(* Logix 5000 project; controller cal1615 1756-L62 rev 20.19; software revision 20.05; part 25 of 81 *)
(* tags used below, declared in another part *)
   FAULT : BOOL;   // Fault AFI
   p01_param_oven_timer_presets : DINT[32];   // System Parameter Oven Timer Presets
   p01_param_process_air_hl : REAL;   // Machine Parameter Process Air High Limit
   p01_sys_lc : Limit_Clamp;   // Zone 1 Misc Control Limit Clamp
   p01r09_pb_global_reset : BOOL;   // System Modes PB: Global Fault Reset
   p01r11 : routine;   // System Timer Presets
   p02_real_from_hmi : hmi_real;   // MOP HMI Iface Real from HMI
   p12_dint_to_hmi : DINT[16];   // Zone 2 Temperature Control VFDs On
   p12_param_fast_to_soak : REAL;   // Zone 2 Parameter Fast to Soak Control
   p12_param_lfl_hhl : REAL;   // Zone 2 Parameter High High Lower Flash Limit
   p12_param_lfl_hl : REAL;   // Zone 2 Parameter High LFL Limit
   p12_param_pid1_ff : REAL;   // Zone 2 Parameter Fast PID Bias
   p12_param_pid1_kd : REAL;   // Zone 2 Parameter Fast PID Derivative Gain
   p12_param_pid1_ki : REAL;   // Zone 2 Parameter Fast PID Integral Gain
   p12_param_pid1_kp : REAL;   // Zone 2 Parameter Fast PID Proportional Gain
   p12_param_pid2_ff : REAL;   // Zone 2 Parameter Auto PID Bias
   p12_param_pid2_kd : REAL;   // Zone 2 Parameter Auto PID Derivative Gain
   p12_param_pid2_ki : REAL;   // Zone 2 Parameter Auto PID Integral Gain
   p12_param_pid2_kp : REAL;   // Zone 2 Parameter Auto PID Proportional Gain
   p12_param_shutdown_temp : REAL;   // Zone 2 Parameter Zone Shutdown Temperature
   p12_param_soak_to_fast : REAL;   // Zone 2 Parameter Soak to Fast Control
   p12_param_tc01_dev : REAL;   // Zone 2 Parameter Oven Temperature Deviation from Setpoint
   p12_param_tc01_hl : REAL;   // Zone 2 Parameter Process Air High Limit
   p12_param_tc01z : REAL;   // Zone 2 Parameter Process Temperature Zero Offset
   p12_param_tc02z : REAL;   // Zone 2 Parameter SupplyTemperature Zero Offset
   p12_param_zone_pressure : REAL;   // Zone 2 Parameter High Pressure LImit
   p12r01 : routine;   // Zone 2 Main
   p12r02 : routine;   // Zone 2 Misc Control
   p12r02_timer_safe_temp : TIMER[2];   // Zone 2 Misc Control Chamber SafeTemperature Dwell
   p12r02_timer_warning : TIMER[4];   // Zone 2 Misc Control Warning Delay
   p12r08 : routine;   // Zone 2 Warnings
   p12r08_timer_fault : TIMER[4];   // Zone 2 Warnings Fault Delay
   p12r08_timer_warning : TIMER[4];   // Zone 2 Warnings Warning Delay
   p12r09 : routine;   // Zone 2 Modes
   p12r09_timer_fault : TIMER[4];   // Zone 2 Modes Fault Delay
   p12r09_timer_warning : TIMER[8];   // Zone 2 Modes Warning Delay
   p12r10 : routine;   // Zone 2
   p12r10_timer_fault : TIMER[4];   // Zone 2 Fault Delay
   p12r10_timer_warning : TIMER[4];   // Zone 2 Warning Delay
   p12r20_timer_state_11 : TIMER;   // Zone 2 Temp Sequence State 11 Dwell
   p12r20_timer_state_3 : TIMER;   // Zone 2 Temperature Control State 3 Dwell
   p12r20_timer_state_4 : TIMER;   // Zone 2 Temp Sequence State 4 Dwell
   p12r20_timer_state_7 : TIMER;   // Zone 2 Temp Sequence State 7 Dwell
   p12r30 : routine;   // Zone 2 Temperature Control
   p12r30_cv_man_sp : REAL;   // Zone 2 Temperature Control Manual Heat Control Valve Setpoint
   p12r30_temp_deviation_setpoint : DINT;
   p12r30_timer_fault : TIMER[16];   // Zone 2 Temperature Control Fault Delay
   p12r30_timer_warning : TIMER[12];   // Zone 2 Temperature Control Warning Delay
   p12r31 : routine;   // Zone 2 Exhaust VFD
   p12r31_timer_fault : TIMER[5];   // Zone 2 Exhaust VFD Fault Timer
   p12r31_timer_warning : TIMER[5];   // Zone 2 Exhaust VFD Waringing Timer
   p12r32 : routine;   // Zone 2 Recirc VFD
   p12r32_timer_fault : TIMER[5];   // Zone 2 Recirc VFD Fault Timer
   p12r32_timer_warning : TIMER[5];   // Zone 2 Supply VFD Warning Timer
(* P12_Zone_2, continued *)

ROUTINE R08_Warnings   (* ladder *)
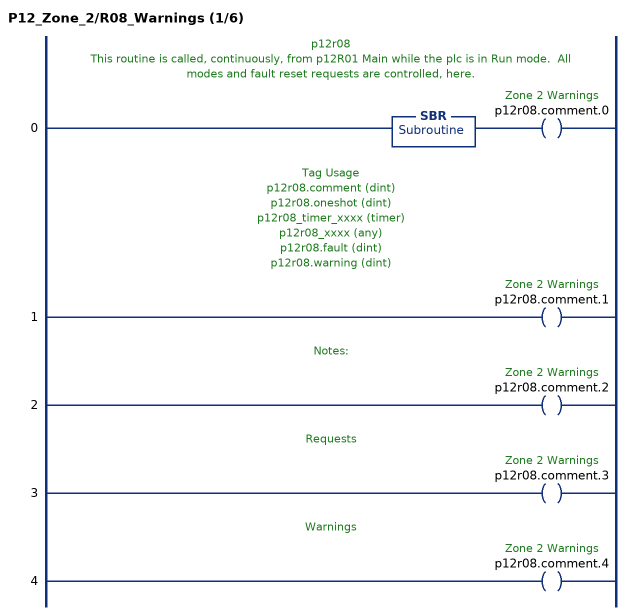
   // p12r08
   // This routine is called, continuously, from p12R01 Main while the plc is in Run mode.  All modes and fault reset requests are controlled, here.
   0: SBR()OTE(p12r08.comment.0);
   // Tag Usage
   // p12r08.comment (dint)
   // p12r08.oneshot (dint)
   // p12r08_timer_xxxx (timer)
   // p12r08_xxxx (any)
   // p12r08.fault (dint)
   // p12r08.warning (dint)
   1: OTE(p12r08.comment.1);
   // Notes:
   2: OTE(p12r08.comment.2);
   // Requests
   3: OTE(p12r08.comment.3);
   // Warnings
   4: OTE(p12r08.comment.4);
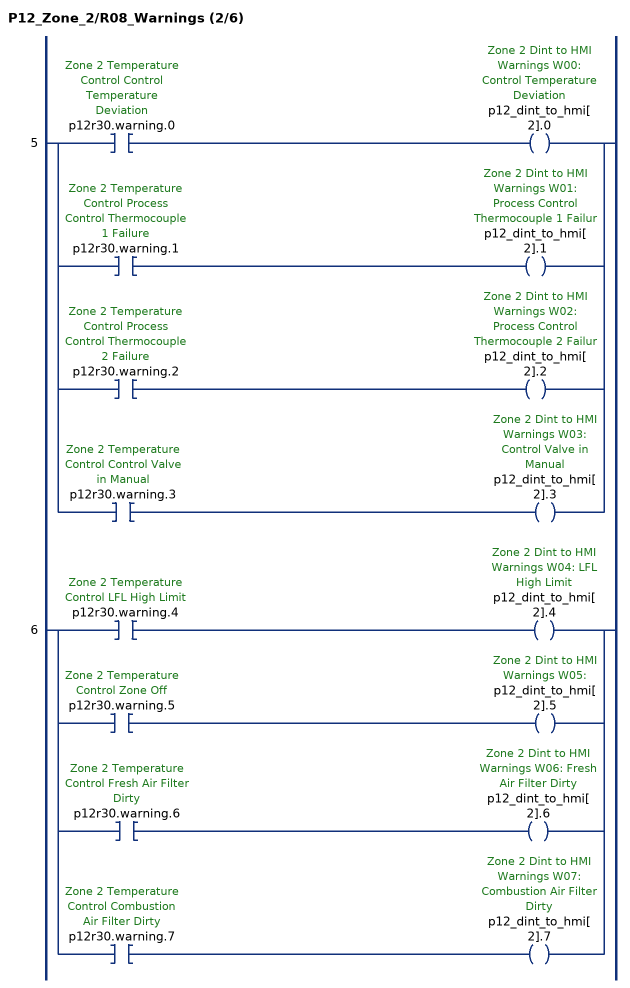
   5: [XIC(p12r30.warning.0) OTE(p12_dint_to_hmi[2].0) ,XIC(p12r30.warning.1) OTE(p12_dint_to_hmi[2].1) ,XIC(p12r30.warning.2) OTE(p12_dint_to_hmi[2].2) ,XIC(p12r30.warning.3) OTE(p12_dint_to_hmi[2].3) ];
   6: [XIC(p12r30.warning.4) OTE(p12_dint_to_hmi[2].4) ,XIC(p12r30.warning.5) OTE(p12_dint_to_hmi[2].5) ,XIC(p12r30.warning.6) OTE(p12_dint_to_hmi[2].6) ,XIC(p12r30.warning.7) OTE(p12_dint_to_hmi[2].7) ];
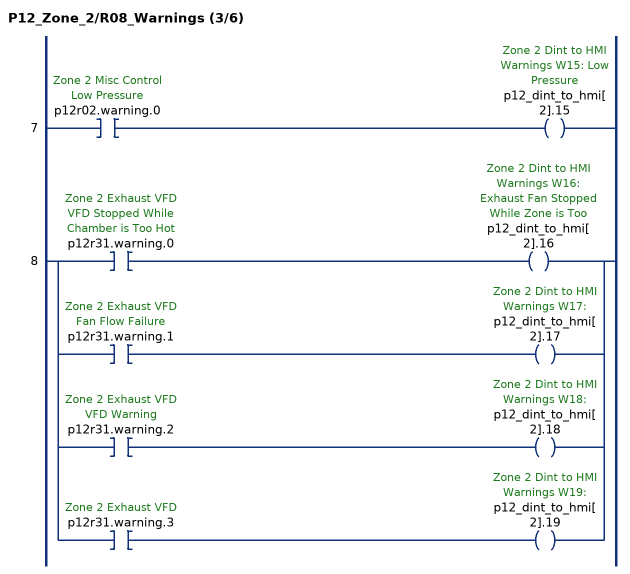
   7: XIC(p12r02.warning.0)OTE(p12_dint_to_hmi[2].15);
   8: [XIC(p12r31.warning.0) OTE(p12_dint_to_hmi[2].16) ,XIC(p12r31.warning.1) OTE(p12_dint_to_hmi[2].17) ,XIC(p12r31.warning.2) OTE(p12_dint_to_hmi[2].18) ,XIC(p12r31.warning.3) OTE(p12_dint_to_hmi[2].19) ];
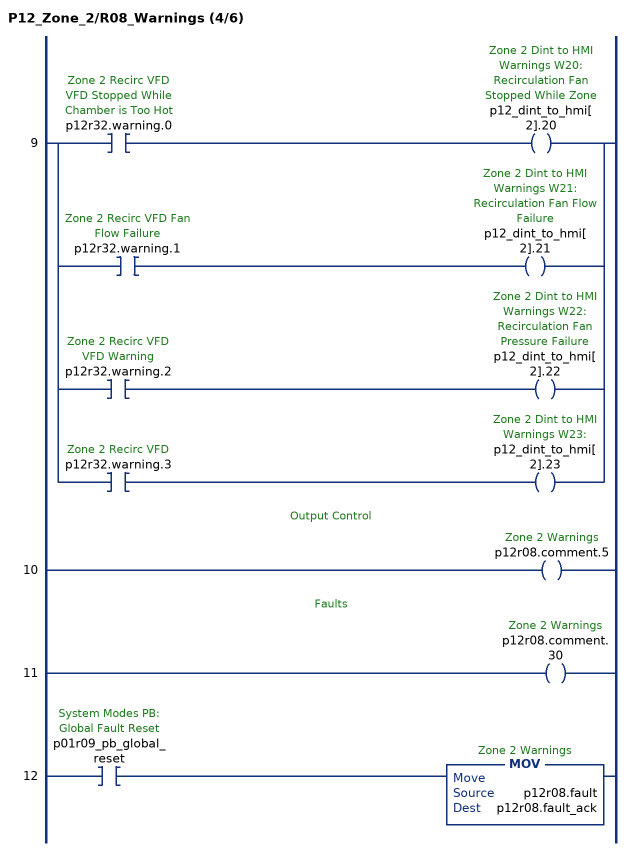
   9: [XIC(p12r32.warning.0) OTE(p12_dint_to_hmi[2].20) ,XIC(p12r32.warning.1) OTE(p12_dint_to_hmi[2].21) ,XIC(p12r32.warning.2) OTE(p12_dint_to_hmi[2].22) ,XIC(p12r32.warning.3) OTE(p12_dint_to_hmi[2].23) ];
   // Output Control
   10: OTE(p12r08.comment.5);
   // Faults
   11: OTE(p12r08.comment.30);
   12: XIC(p01r09_pb_global_reset)MOV(p12r08.fault,p12r08.fault_ack);
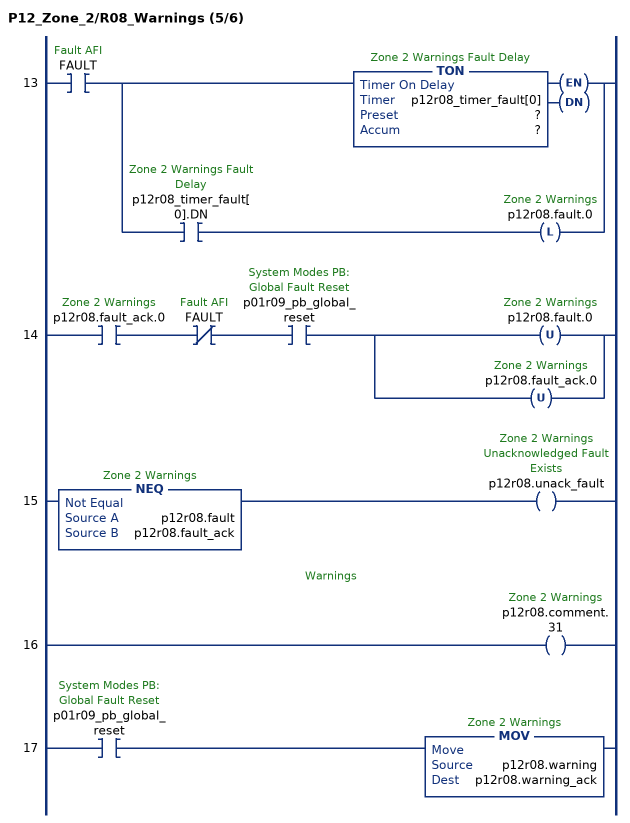
   13: XIC(FAULT)[TON(p12r08_timer_fault[0],?,?) ,XIC(p12r08_timer_fault[0].DN) OTL(p12r08.fault.0) ];
   14: XIC(p12r08.fault_ack.0)XIO(FAULT)XIC(p01r09_pb_global_reset)[OTU(p12r08.fault.0) ,OTU(p12r08.fault_ack.0) ];
   15: NEQ(p12r08.fault,p12r08.fault_ack)OTE(p12r08.unack_fault);
   // Warnings
   16: OTE(p12r08.comment.31);
   17: XIC(p01r09_pb_global_reset)MOV(p12r08.warning,p12r08.warning_ack);
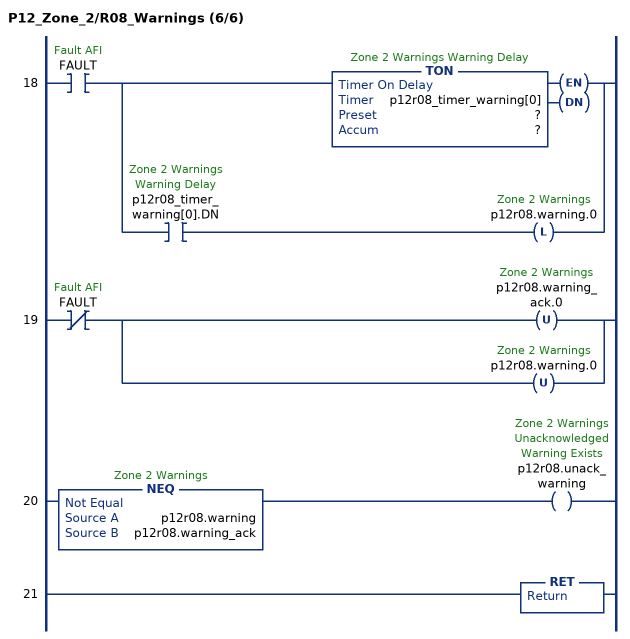
   18: XIC(FAULT)[TON(p12r08_timer_warning[0],?,?) ,XIC(p12r08_timer_warning[0].DN) OTL(p12r08.warning.0) ];
   19: XIO(FAULT)[OTU(p12r08.warning_ack.0) ,OTU(p12r08.warning.0) ];
   20: NEQ(p12r08.warning,p12r08.warning_ack)OTE(p12r08.unack_warning);
   21: RET();
END_ROUTINE

ROUTINE R09_Modes   (* ladder *)
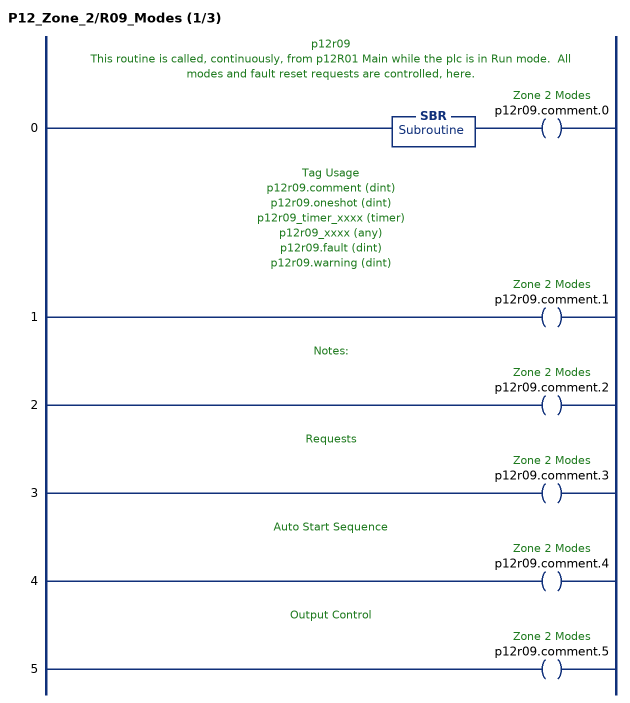
   // p12r09
   // This routine is called, continuously, from p12R01 Main while the plc is in Run mode.  All modes and fault reset requests are controlled, here.
   0: SBR()OTE(p12r09.comment.0);
   // Tag Usage
   // p12r09.comment (dint)
   // p12r09.oneshot (dint)
   // p12r09_timer_xxxx (timer)
   // p12r09_xxxx (any)
   // p12r09.fault (dint)
   // p12r09.warning (dint)
   1: OTE(p12r09.comment.1);
   // Notes:
   2: OTE(p12r09.comment.2);
   // Requests
   3: OTE(p12r09.comment.3);
   // Auto Start Sequence
   4: OTE(p12r09.comment.4);
   // Output Control
   5: OTE(p12r09.comment.5);
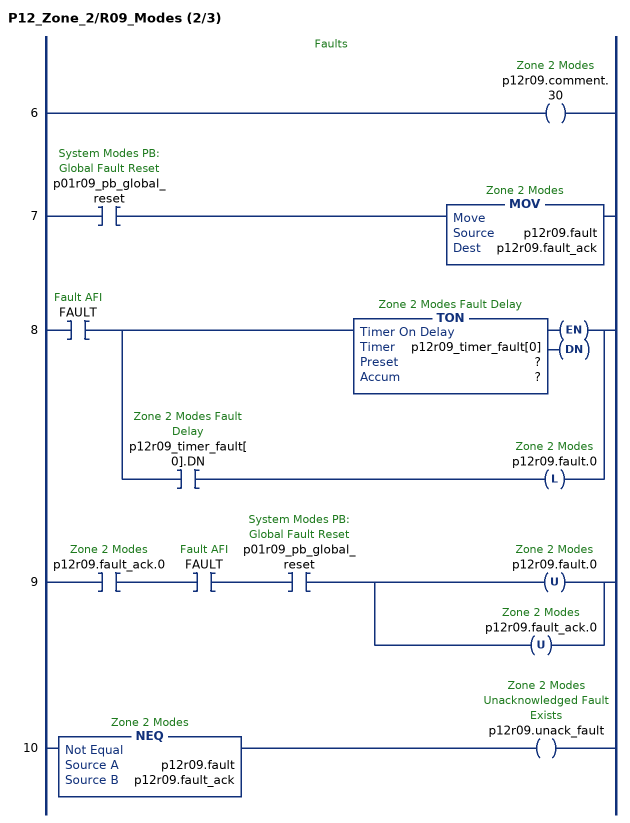
   // Faults
   6: OTE(p12r09.comment.30);
   7: XIC(p01r09_pb_global_reset)MOV(p12r09.fault,p12r09.fault_ack);
   8: XIC(FAULT)[TON(p12r09_timer_fault[0],?,?) ,XIC(p12r09_timer_fault[0].DN) OTL(p12r09.fault.0) ];
   9: XIC(p12r09.fault_ack.0)XIC(FAULT)XIC(p01r09_pb_global_reset)[OTU(p12r09.fault.0) ,OTU(p12r09.fault_ack.0) ];
   10: NEQ(p12r09.fault,p12r09.fault_ack)OTE(p12r09.unack_fault);
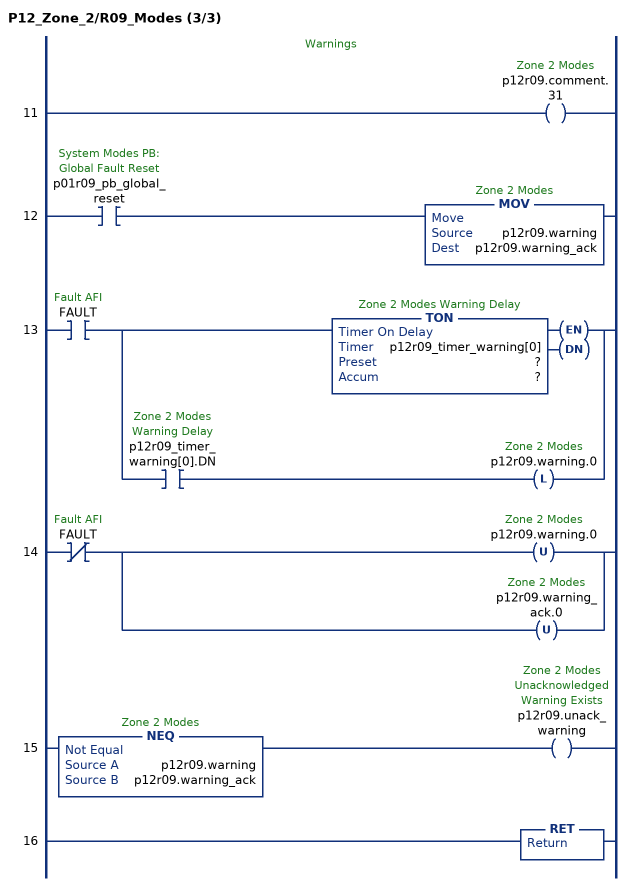
   // Warnings
   11: OTE(p12r09.comment.31);
   12: XIC(p01r09_pb_global_reset)MOV(p12r09.warning,p12r09.warning_ack);
   13: XIC(FAULT)[TON(p12r09_timer_warning[0],?,?) ,XIC(p12r09_timer_warning[0].DN) OTL(p12r09.warning.0) ];
   14: XIO(FAULT)[OTU(p12r09.warning.0) ,OTU(p12r09.warning_ack.0) ];
   15: NEQ(p12r09.warning,p12r09.warning_ack)OTE(p12r09.unack_warning);
   16: RET();
END_ROUTINE

ROUTINE R10_Parameters   (* ladder *)
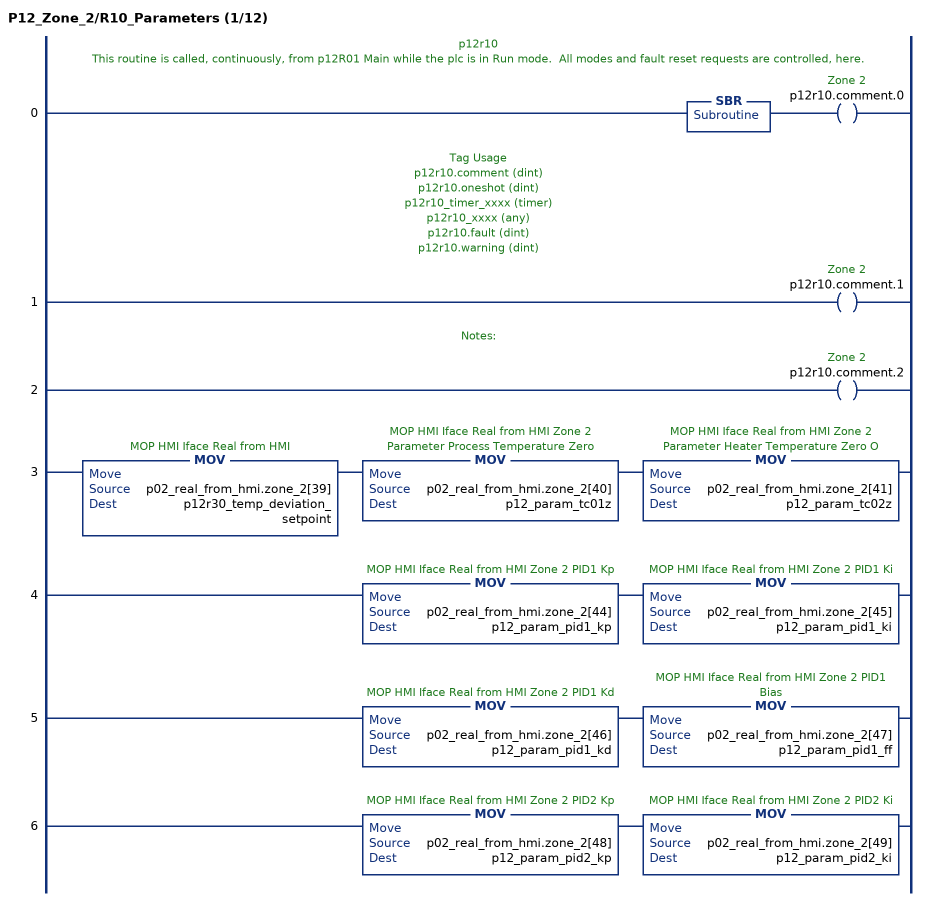
   // p12r10
   // This routine is called, continuously, from p12R01 Main while the plc is in Run mode.  All modes and fault reset requests are controlled, here.
   0: SBR()OTE(p12r10.comment.0);
   // Tag Usage
   // p12r10.comment (dint)
   // p12r10.oneshot (dint)
   // p12r10_timer_xxxx (timer)
   // p12r10_xxxx (any)
   // p12r10.fault (dint)
   // p12r10.warning (dint)
   1: OTE(p12r10.comment.1);
   // Notes:
   2: OTE(p12r10.comment.2);
   3: MOV(p02_real_from_hmi.zone_2[39],p12r30_temp_deviation_setpoint)MOV(p02_real_from_hmi.zone_2[40],p12_param_tc01z)MOV(p02_real_from_hmi.zone_2[41],p12_param_tc02z);
   4: MOV(p02_real_from_hmi.zone_2[44],p12_param_pid1_kp)MOV(p02_real_from_hmi.zone_2[45],p12_param_pid1_ki);
   5: MOV(p02_real_from_hmi.zone_2[46],p12_param_pid1_kd)MOV(p02_real_from_hmi.zone_2[47],p12_param_pid1_ff);
   6: MOV(p02_real_from_hmi.zone_2[48],p12_param_pid2_kp)MOV(p02_real_from_hmi.zone_2[49],p12_param_pid2_ki);
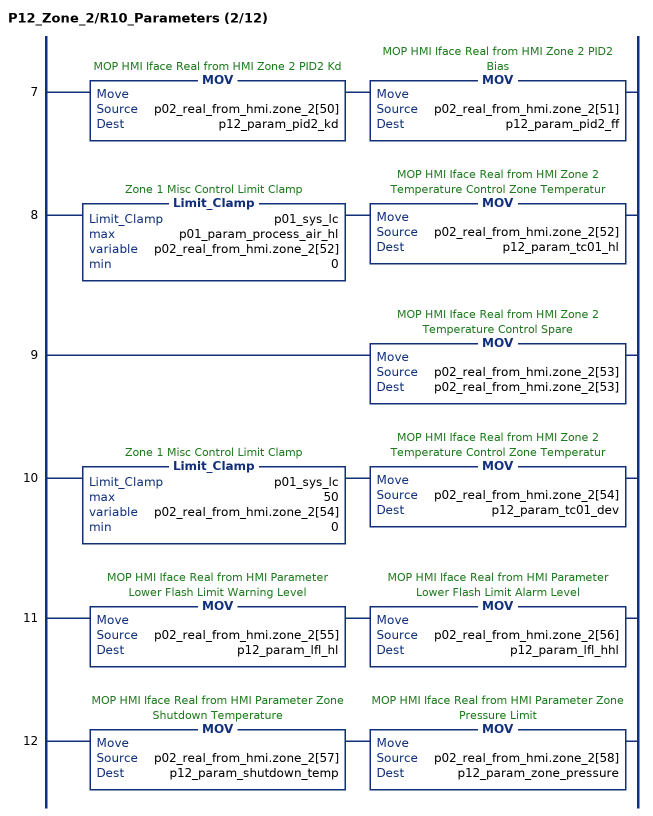
   7: MOV(p02_real_from_hmi.zone_2[50],p12_param_pid2_kd)MOV(p02_real_from_hmi.zone_2[51],p12_param_pid2_ff);
   8: Limit_Clamp(p01_sys_lc,p01_param_process_air_hl,p02_real_from_hmi.zone_2[52],0)MOV(p02_real_from_hmi.zone_2[52],p12_param_tc01_hl);
   9: MOV(p02_real_from_hmi.zone_2[53],p02_real_from_hmi.zone_2[53]);
   10: Limit_Clamp(p01_sys_lc,50,p02_real_from_hmi.zone_2[54],0)MOV(p02_real_from_hmi.zone_2[54],p12_param_tc01_dev);
   11: MOV(p02_real_from_hmi.zone_2[55],p12_param_lfl_hl)MOV(p02_real_from_hmi.zone_2[56],p12_param_lfl_hhl);
   12: MOV(p02_real_from_hmi.zone_2[57],p12_param_shutdown_temp)MOV(p02_real_from_hmi.zone_2[58],p12_param_zone_pressure);
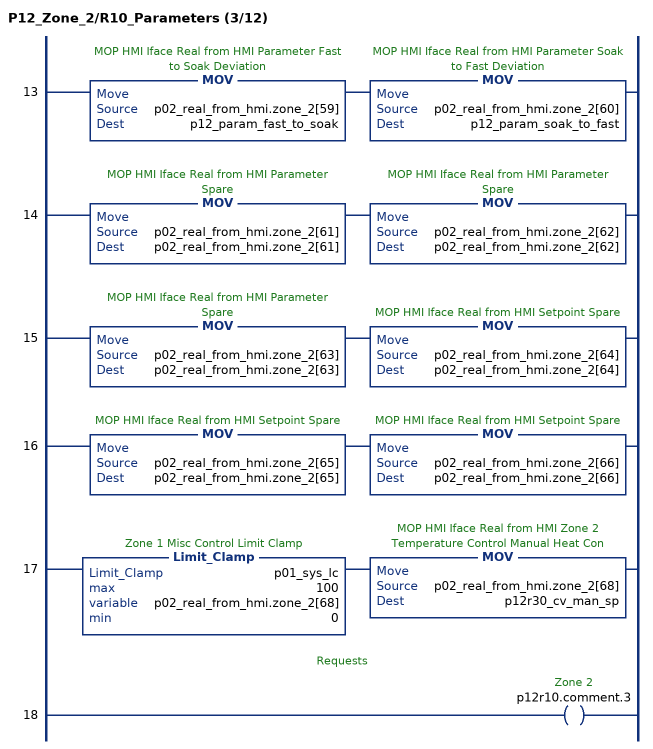
   13: MOV(p02_real_from_hmi.zone_2[59],p12_param_fast_to_soak)MOV(p02_real_from_hmi.zone_2[60],p12_param_soak_to_fast);
   14: MOV(p02_real_from_hmi.zone_2[61],p02_real_from_hmi.zone_2[61])MOV(p02_real_from_hmi.zone_2[62],p02_real_from_hmi.zone_2[62]);
   15: MOV(p02_real_from_hmi.zone_2[63],p02_real_from_hmi.zone_2[63])MOV(p02_real_from_hmi.zone_2[64],p02_real_from_hmi.zone_2[64]);
   16: MOV(p02_real_from_hmi.zone_2[65],p02_real_from_hmi.zone_2[65])MOV(p02_real_from_hmi.zone_2[66],p02_real_from_hmi.zone_2[66]);
   17: Limit_Clamp(p01_sys_lc,100,p02_real_from_hmi.zone_2[68],0)MOV(p02_real_from_hmi.zone_2[68],p12r30_cv_man_sp);
   // Requests
   18: OTE(p12r10.comment.3);
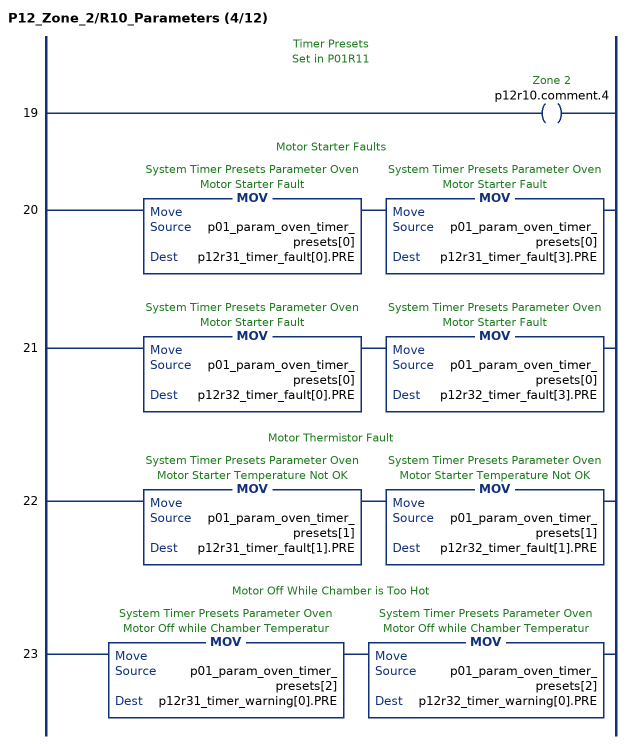
   // Timer Presets
   // Set in P01R11
   19: OTE(p12r10.comment.4);
   // Motor Starter Faults
   20: MOV(p01_param_oven_timer_presets[0],p12r31_timer_fault[0].PRE)MOV(p01_param_oven_timer_presets[0],p12r31_timer_fault[3].PRE);
   21: MOV(p01_param_oven_timer_presets[0],p12r32_timer_fault[0].PRE)MOV(p01_param_oven_timer_presets[0],p12r32_timer_fault[3].PRE);
   // Motor Thermistor Fault
   22: MOV(p01_param_oven_timer_presets[1],p12r31_timer_fault[1].PRE)MOV(p01_param_oven_timer_presets[1],p12r32_timer_fault[1].PRE);
   // Motor Off While Chamber is Too Hot
   23: MOV(p01_param_oven_timer_presets[2],p12r31_timer_warning[0].PRE)MOV(p01_param_oven_timer_presets[2],p12r32_timer_warning[0].PRE);
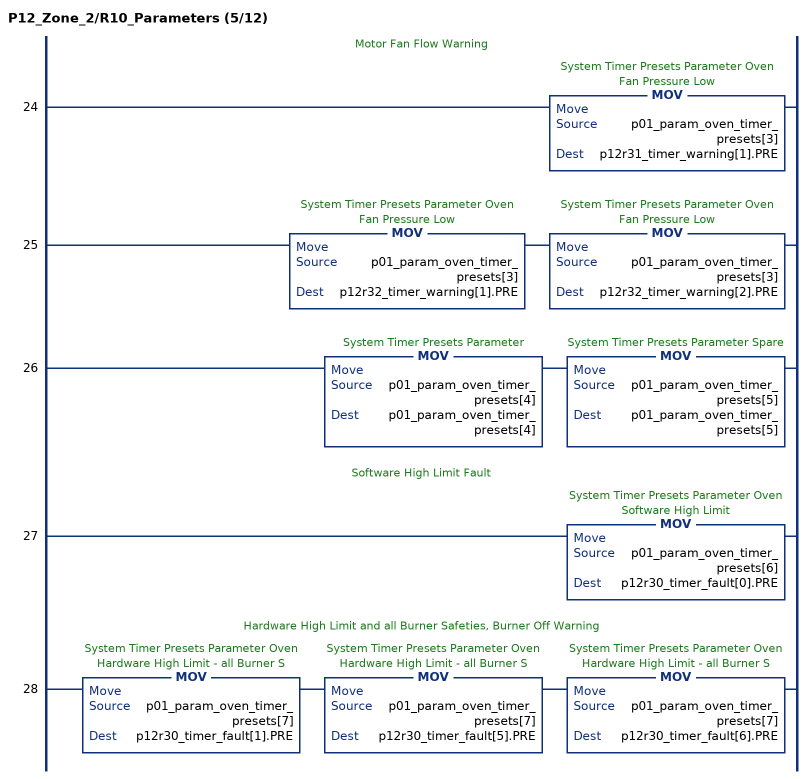
   // Motor Fan Flow Warning
   24: MOV(p01_param_oven_timer_presets[3],p12r31_timer_warning[1].PRE);
   25: MOV(p01_param_oven_timer_presets[3],p12r32_timer_warning[1].PRE)MOV(p01_param_oven_timer_presets[3],p12r32_timer_warning[2].PRE);
   26: MOV(p01_param_oven_timer_presets[4],p01_param_oven_timer_presets[4])MOV(p01_param_oven_timer_presets[5],p01_param_oven_timer_presets[5]);
   // Software High Limit Fault
   27: MOV(p01_param_oven_timer_presets[6],p12r30_timer_fault[0].PRE);
   // Hardware High Limit and all Burner Safeties, Burner Off Warning
   28: MOV(p01_param_oven_timer_presets[7],p12r30_timer_fault[1].PRE)MOV(p01_param_oven_timer_presets[7],p12r30_timer_fault[5].PRE)MOV(p01_param_oven_timer_presets[7],p12r30_timer_fault[6].PRE);
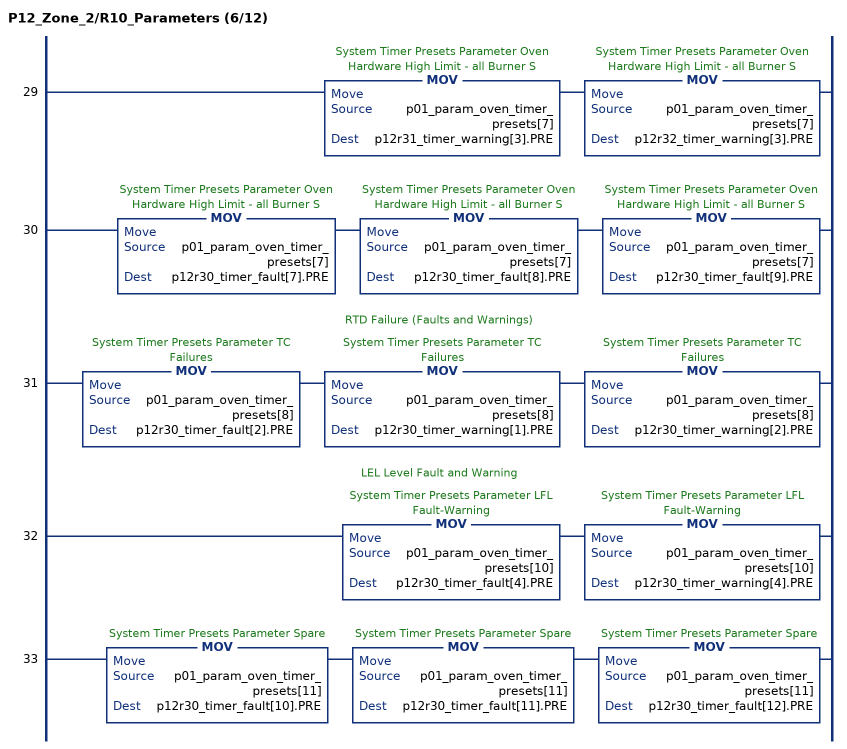
   29: MOV(p01_param_oven_timer_presets[7],p12r31_timer_warning[3].PRE)MOV(p01_param_oven_timer_presets[7],p12r32_timer_warning[3].PRE);
   30: MOV(p01_param_oven_timer_presets[7],p12r30_timer_fault[7].PRE)MOV(p01_param_oven_timer_presets[7],p12r30_timer_fault[8].PRE)MOV(p01_param_oven_timer_presets[7],p12r30_timer_fault[9].PRE);
   // RTD Failure (Faults and Warnings)
   31: MOV(p01_param_oven_timer_presets[8],p12r30_timer_fault[2].PRE)MOV(p01_param_oven_timer_presets[8],p12r30_timer_warning[1].PRE)MOV(p01_param_oven_timer_presets[8],p12r30_timer_warning[2].PRE);
   // LEL Level Fault and Warning
   32: MOV(p01_param_oven_timer_presets[10],p12r30_timer_fault[4].PRE)MOV(p01_param_oven_timer_presets[10],p12r30_timer_warning[4].PRE);
   33: MOV(p01_param_oven_timer_presets[11],p12r30_timer_fault[10].PRE)MOV(p01_param_oven_timer_presets[11],p12r30_timer_fault[11].PRE)MOV(p01_param_oven_timer_presets[11],p12r30_timer_fault[12].PRE);
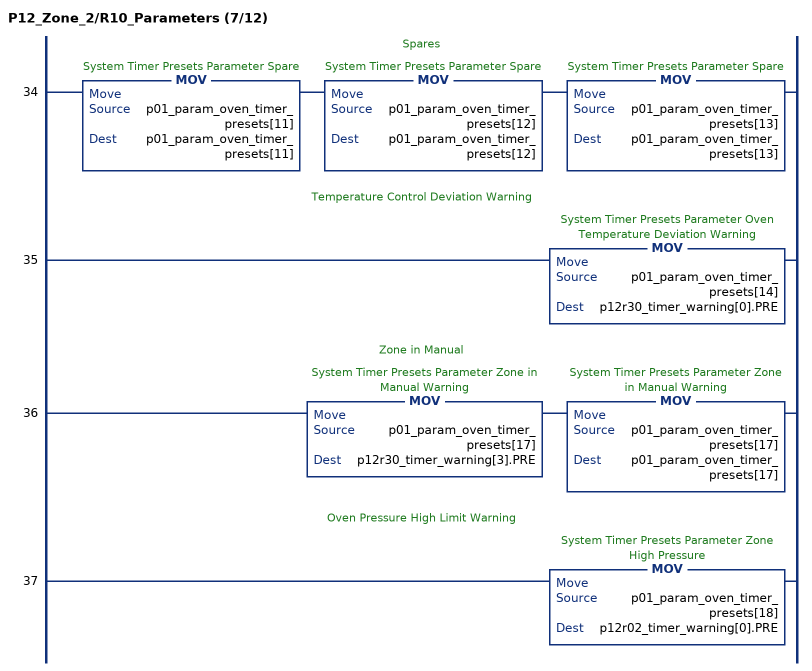
   // Spares
   34: MOV(p01_param_oven_timer_presets[11],p01_param_oven_timer_presets[11])MOV(p01_param_oven_timer_presets[12],p01_param_oven_timer_presets[12])MOV(p01_param_oven_timer_presets[13],p01_param_oven_timer_presets[13]);
   // Temperature Control Deviation Warning
   35: MOV(p01_param_oven_timer_presets[14],p12r30_timer_warning[0].PRE);
   // Zone in Manual
   36: MOV(p01_param_oven_timer_presets[17],p12r30_timer_warning[3].PRE)MOV(p01_param_oven_timer_presets[17],p01_param_oven_timer_presets[17]);
   // Oven Pressure High Limit Warning
   37: MOV(p01_param_oven_timer_presets[18],p12r02_timer_warning[0].PRE);
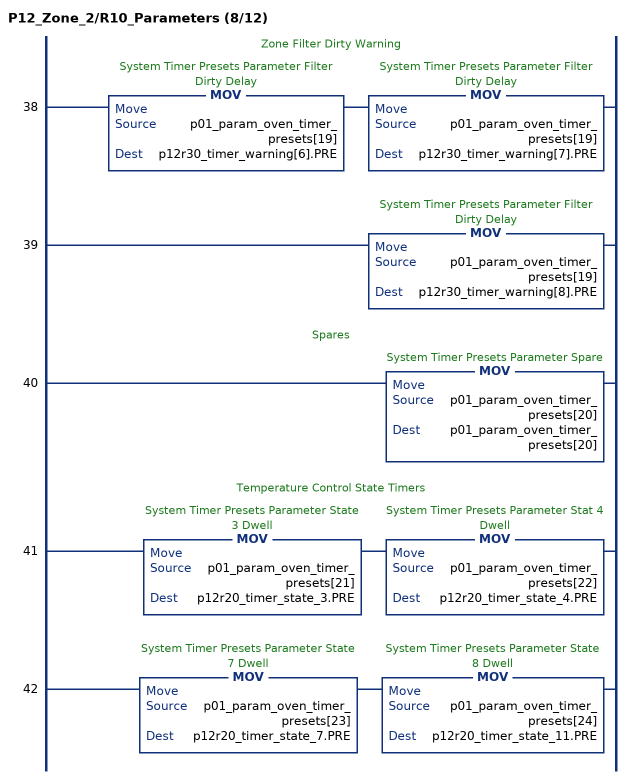
   // Zone Filter Dirty Warning
   38: MOV(p01_param_oven_timer_presets[19],p12r30_timer_warning[6].PRE)MOV(p01_param_oven_timer_presets[19],p12r30_timer_warning[7].PRE);
   39: MOV(p01_param_oven_timer_presets[19],p12r30_timer_warning[8].PRE);
   // Spares
   40: MOV(p01_param_oven_timer_presets[20],p01_param_oven_timer_presets[20]);
   // Temperature Control State Timers
   41: MOV(p01_param_oven_timer_presets[21],p12r20_timer_state_3.PRE)MOV(p01_param_oven_timer_presets[22],p12r20_timer_state_4.PRE);
   42: MOV(p01_param_oven_timer_presets[23],p12r20_timer_state_7.PRE)MOV(p01_param_oven_timer_presets[24],p12r20_timer_state_11.PRE);
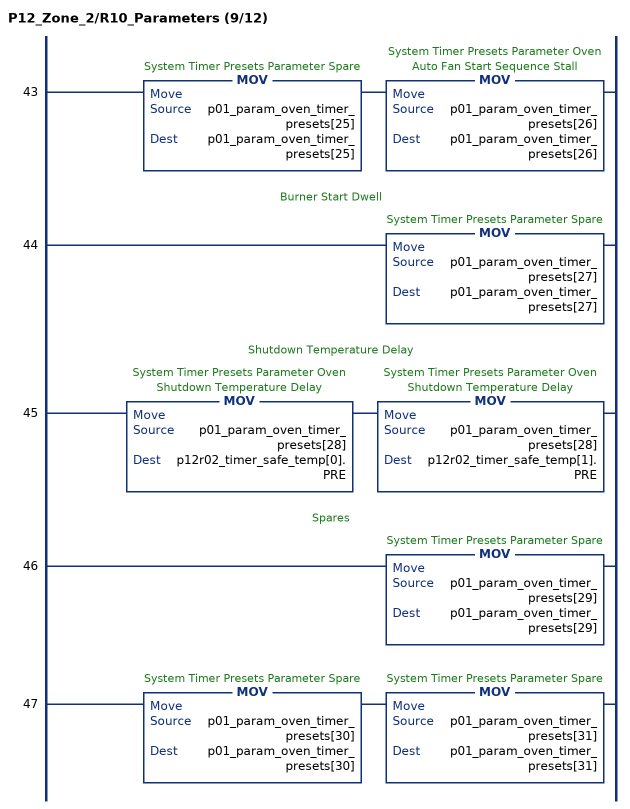
   43: MOV(p01_param_oven_timer_presets[25],p01_param_oven_timer_presets[25])MOV(p01_param_oven_timer_presets[26],p01_param_oven_timer_presets[26]);
   // Burner Start Dwell
   44: MOV(p01_param_oven_timer_presets[27],p01_param_oven_timer_presets[27]);
   // Shutdown Temperature Delay
   45: MOV(p01_param_oven_timer_presets[28],p12r02_timer_safe_temp[0].PRE)MOV(p01_param_oven_timer_presets[28],p12r02_timer_safe_temp[1].PRE);
   // Spares
   46: MOV(p01_param_oven_timer_presets[29],p01_param_oven_timer_presets[29]);
   47: MOV(p01_param_oven_timer_presets[30],p01_param_oven_timer_presets[30])MOV(p01_param_oven_timer_presets[31],p01_param_oven_timer_presets[31]);
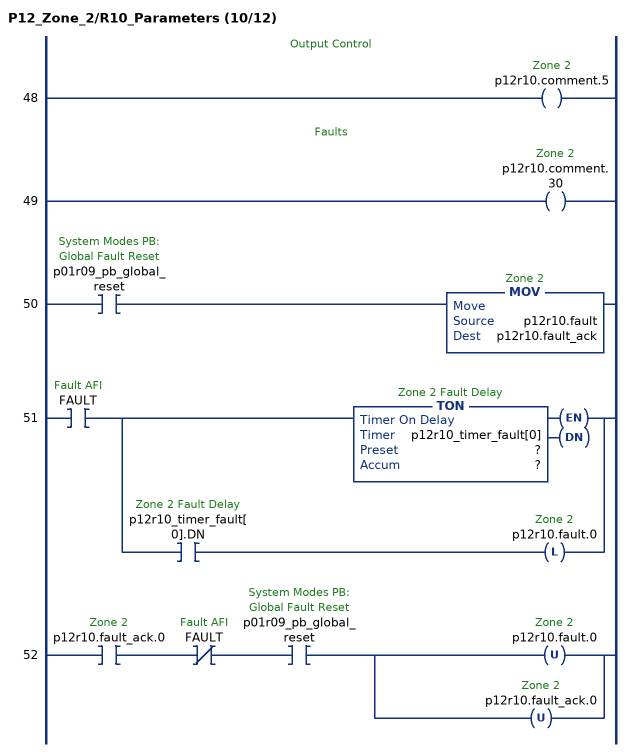
   // Output Control
   48: OTE(p12r10.comment.5);
   // Faults
   49: OTE(p12r10.comment.30);
   50: XIC(p01r09_pb_global_reset)MOV(p12r10.fault,p12r10.fault_ack);
   51: XIC(FAULT)[TON(p12r10_timer_fault[0],?,?) ,XIC(p12r10_timer_fault[0].DN) OTL(p12r10.fault.0) ];
   52: XIC(p12r10.fault_ack.0)XIO(FAULT)XIC(p01r09_pb_global_reset)[OTU(p12r10.fault.0) ,OTU(p12r10.fault_ack.0) ];
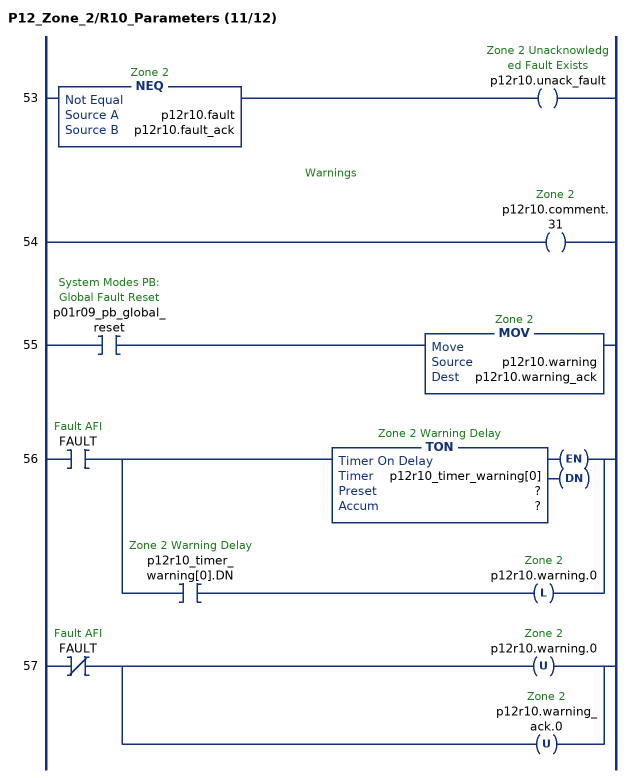
   53: NEQ(p12r10.fault,p12r10.fault_ack)OTE(p12r10.unack_fault);
   // Warnings
   54: OTE(p12r10.comment.31);
   55: XIC(p01r09_pb_global_reset)MOV(p12r10.warning,p12r10.warning_ack);
   56: XIC(FAULT)[TON(p12r10_timer_warning[0],?,?) ,XIC(p12r10_timer_warning[0].DN) OTL(p12r10.warning.0) ];
   57: XIO(FAULT)[OTU(p12r10.warning.0) ,OTU(p12r10.warning_ack.0) ];
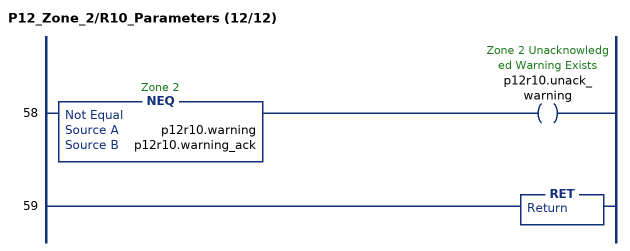
   58: NEQ(p12r10.warning,p12r10.warning_ack)OTE(p12r10.unack_warning);
   59: RET();
END_ROUTINE
